FUNCTION "ChangeOverProcess" : Void
VAR_TEMP
  tBool : Bool;
END_VAR
BEGIN
  // Původní jazyk: LAD
  // Zdroj XML: EXPORT/Program blocks/OP010/03_Auto/01ChangeOver/ChangeOverProcess.xml
  // (Žádný StructuredText network nebyl nalezen; LAD/STL/GRAPH není automaticky překládán.)
END_FUNCTION
